FUNCTION TryConvert_TOD_TO_SINT : BOOL
VAR_INPUT
	in : TOD;
	out : REFERENCE TO SINT;
END_VAR

IF in > DatatypeLimits.MAX_VALUE_OF_TOD_WHICH_CAN_BE_HELD_IN_A_SINT THEN
	RETURN;
END_IF

out := TOD_TO_SINT(in);
TryConvert_TOD_TO_SINT := TRUE;

END_FUNCTION

(* stored: Version 1.1.0.1, ProductVersion 3.1.4024.12
   POU TryConvert_TOD_TO_SINT: Id {1fcac14b-5f32-41ca-9604-b3fb765816a3}, SpecialFunc None *)
